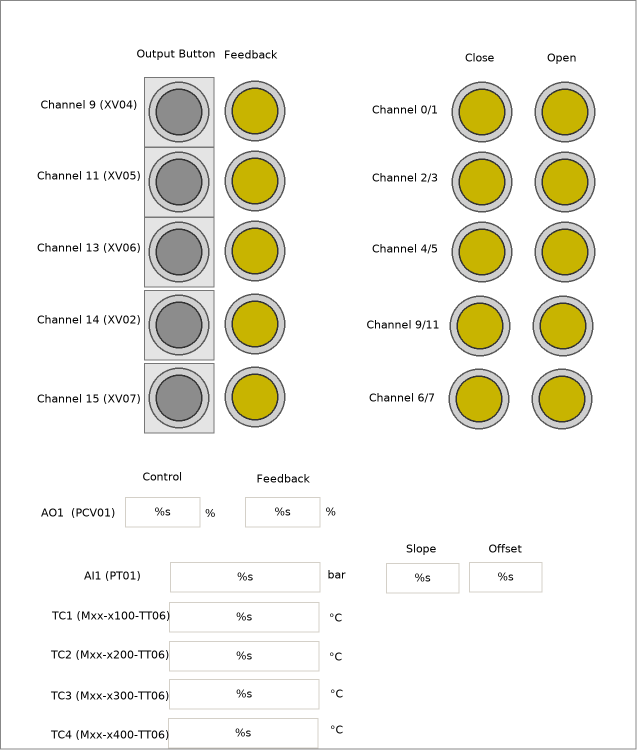
VISUALIZATION rs1  // 637x750
    Lamp1 (220,289 70x70), variable: bDigitalOutFdbk[4], style: Lamp-Lamp1-Yellow
    PushSwitch (144,290 70x70), variable: bDigitalOut[4], behaviour: TOGGLE, style: Switch-PushSwitch-Gray
    PushSwitch (144,77 70x70), variable: bDigitalOut[1], behaviour: TOGGLE, style: Switch-PushSwitch-Gray
    PushSwitch (144,147 70x70), variable: bDigitalOut[2], behaviour: TOGGLE, style: Switch-PushSwitch-Gray
    PushSwitch (144,217 70x70), variable: bDigitalOut[3], behaviour: TOGGLE, style: Switch-PushSwitch-Gray
    PushSwitch (144,363 70x70), variable: bDigitalOut[5], behaviour: TOGGLE, style: Switch-PushSwitch-Gray
    Lamp1 (220,76 70x70), variable: bDigitalOutFdbk[1], style: Lamp-Lamp1-Yellow
    Lamp1 (220,146 70x70), variable: bDigitalOutFdbk[2], style: Lamp-Lamp1-Yellow
    Lamp1 (220,216 70x70), variable: bDigitalOutFdbk[3], style: Lamp-Lamp1-Yellow
    Lamp1 (220,362 70x70), variable: bDigitalOutFdbk[5], style: Lamp-Lamp1-Yellow
    Label (101,39 150x30), "Output Button"
    Label (176,40 150x30), "Feedback"
    Label (14,305 150x30), "Channel 14 (XV02)"
    Label (14,90 150x30), "Channel 9 (XV04)"
    Label (14,161 150x30), "Channel 11 (XV05)"
    Label (14,233 150x30), "Channel 13 (XV06)"
    Label (14,384 150x30), "Channel 15 (XV07)"
    Lamp1 (447,77 70x70), variable: GVL_DigitalIn.bDigitalIn[1], style: Lamp-Lamp1-Yellow
    Lamp1 (530,77 70x70), variable: GVL_DigitalIn.bDigitalIn[2], style: Lamp-Lamp1-Yellow
    Lamp1 (447,147 70x70), variable: GVL_DigitalIn.bDigitalIn[3], style: Lamp-Lamp1-Yellow
    Lamp1 (530,147 70x70), variable: GVL_DigitalIn.bDigitalIn[4], style: Lamp-Lamp1-Yellow
    Lamp1 (447,217 70x70), variable: GVL_DigitalIn.bDigitalIn[5], style: Lamp-Lamp1-Yellow
    Lamp1 (530,217 70x70), variable: GVL_DigitalIn.bDigitalIn[6], style: Lamp-Lamp1-Yellow
    Lamp1 (444,364 70x70), variable: GVL_DigitalIn.bDigitalIn[7], style: Lamp-Lamp1-Yellow
    Lamp1 (527,364 70x70), variable: GVL_DigitalIn.bDigitalIn[8], style: Lamp-Lamp1-Yellow
    Label (330,95 150x30), "Channel 0/1"
    Label (330,163 150x30), "Channel 2/3"
    Label (330,234 150x30), "Channel 4/5"
    Label (327,383 150x30), "Channel 6/7"
    Textfield (169,602 150x30), "%s", text variable: GVL_Thermocouples.hmi_config[1].rTempC
    Label (36,601 151x30), "TC1 (Mxx-x100-TT06)"
    Textfield (169,641 150x30), "%s", text variable: GVL_Thermocouples.hmi_config[2].rTempC
    Textfield (169,679 150x30), "%s", text variable: GVL_Thermocouples.hmi_config[3].rTempC
    Textfield (168,718 150x30), "%s", text variable: GVL_Thermocouples.hmi_config[4].rTempC
    Label (405,43 150x30), "Close"
    Label (487,43 150x30), "Open"
    Label (35,640 151x30), "TC2 (Mxx-x200-TT06)"
    Label (35,681 151x30), "TC3 (Mxx-x300-TT06)"
    Label (35,720 151x30), "TC4 (Mxx-x400-TT06)"
    Textfield (125,497 75x30), "%s", text variable: GVL_AnalogOutputs.in_cmd[1]
        OnMouseDown: write the text variable via Default
    Label (3,498 151x30), "AO1 (PCV01)"
    Label (195,498 31x31), "%"
    Textfield (245,497 75x30), "%s", text variable: GVL_AnalogOutputs.fdbk[1]
    Label (316,497 30x30), "%"
    Label (208,464 151x30), "Feedback"
    Label (87,462 151x30), "Control"
    Label (260,603 151x30), "°C"
    Label (260,642 151x30), "°C"
    Label (261,679 151x30), "°C"
    Label (261,715 151x30), "°C"
    Textfield (170,562 150x30), "%s", text variable: GVL_AnalogInputs.hmi_config[1].rEngUnit
    Label (37,561 151x30), "AI1 (PT01)"
    Label (313,560 47x30), "bar"
    Textfield (386,563 73x30), "%s", text variable: GVL_AnalogInputs.hmi_config[1].slope
        OnMouseDown: write the text variable via Default
    Textfield (469,562 73x30), "%s", text variable: GVL_AnalogInputs.hmi_config[1].offset
        OnMouseDown: write the text variable via Default
    Label (384,534 75x30), "Slope"
    Label (468,534 75x30), "Offset"
    Lamp1 (445,291 70x70), variable: GVL_DigitalIn.bDigitalIn[9], style: Lamp-Lamp1-Yellow
    Lamp1 (528,291 70x70), variable: GVL_DigitalIn.bDigitalIn[10], style: Lamp-Lamp1-Yellow
    Label (328,310 150x30), "Channel 9/11"
END_VISUALIZATION

(* stored: Version 1.1.0.1, ProductVersion 3.1.4024.12
   Visu rs1: Id {11cd67df-a7d4-4459-89e3-b362ec809706} *)
